// TIA Portal V18 export
VAR_GLOBAL   // PLC tag table "Andony"
   Andon1_greenBtn AT %I0.0 : Bool;
   Andon1_yellowBtn AT %I0.1 : Bool;
   Andon1_redBtn AT %I0.2 : Bool;
   Andon1_greenLed AT %Q0.0 : Bool;
   Andon1_yellowLed AT %Q0.1 : Bool;
   Andon1_redLed AT %Q0.2 : Bool;
   Andon2_greenBtn AT %I1.4 : Bool;
   Andon2_yellowBtn AT %I1.5 : Bool;
   Andon2_redBtn AT %I1.6 : Bool;
   Andon2_greenLed AT %Q1.4 : Bool;
   Andon2_yellowLed AT %Q1.5 : Bool;
   Andon2_redLed AT %Q1.6 : Bool;
   Andon3_greenBtn AT %I1.0 : Bool;
   Andon3_yellowBtn AT %I1.1 : Bool;
   Andon3_redBtn AT %I1.2 : Bool;
   Andon3_greenLed AT %Q1.0 : Bool;
   Andon3_yellowLed AT %Q1.1 : Bool;
   Andon3_redLed AT %Q1.2 : Bool;
   Andon4_greenBtn AT %I2.4 : Bool;
   Andon4_yellowBtn AT %I2.5 : Bool;
   Andon4_redBtn AT %I2.6 : Bool;
   Andon4_greenLed AT %Q2.4 : Bool;
   Andon4_yellowLed AT %Q2.5 : Bool;
   Andon4_redLed AT %Q2.6 : Bool;
   Andon5_greenBtn AT %I2.0 : Bool;
   Andon5_yellowBtn AT %I2.1 : Bool;
   Andon5_redBtn AT %I2.2 : Bool;
   Andon5_greenLed AT %Q2.0 : Bool;
   Andon5_yellowLed AT %Q2.1 : Bool;
   Andon5_redLed AT %Q2.2 : Bool;
   Andon6_greenBtn AT %I3.4 : Bool;
   Andon6_yellowBtn AT %I3.5 : Bool;
   Andon6_redBtn AT %I3.6 : Bool;
   Andon6_greenLed AT %Q3.4 : Bool;
   Andon6_yellowLed AT %Q3.5 : Bool;
   Andon6_redLed AT %Q3.6 : Bool;
   Andon7_greenBtn AT %I3.0 : Bool;
   Andon7_yellowBtn AT %I3.1 : Bool;
   Andon7_redBtn AT %I3.2 : Bool;
   Andon7_greenLed AT %Q3.0 : Bool;
   Andon7_yellowLed AT %Q3.1 : Bool;
   Andon7_redLed AT %Q3.2 : Bool;
END_VAR
